(* IEC 61131-3 sources: xPLCCore/codesys_code/Application/APPs/AxisGroupSM (part 3) *)

(* ---- ProcessFlyEventsAndIo.st ---- *)
(* =========== IMPLEMENTATION =========== *)
// 2026-06-23 cleanup: trigger-arm + TTL boilerplate factored into
// ArmFiredTrigger() / TickTtl() helpers; pFly aliases the current slot
// once per iteration so the body reads `pFly^.X` instead of
// `FlyEventBuffer[Index].X` 20-odd times.
TriggerActive := FALSE;
FlyEventAvailableCount := 0;

FOR Index := 0 TO TO_INT(FlyEventBufferSize - 1) DO
    pFly := ADR(FlyEventBuffer[Index]);
    TriggerActive := FALSE;
    TriggerErrorCode := 0;

    CASE pFly^.TriggerType OF
        FlyEventTriggerType.DistanceTrigger:
            // Trigger by Cartesian distance from a fixed WCS point. Uses
            // squared distance to avoid SQRT on every scan. ReadPosition is
            // refreshed by UpdateAxisGroupState earlier in the same scan
            // (AxisGroupSM.st:346) so it's the actual TCP pose for this tick.
            DistDx := ReadPosition.c.x - pFly^.TargetPos_X;
            DistDy := ReadPosition.c.y - pFly^.TargetPos_Y;
            DistDz := ReadPosition.c.z - pFly^.TargetPos_Z;
            DistSq := DistDx*DistDx + DistDy*DistDy + DistDz*DistDz;
            DistThresholdSq := pFly^.TargetDistance * pFly^.TargetDistance;
            // TriggerInBoundary=TRUE: fire on entering the ball (dist <= radius).
            // TriggerInBoundary=FALSE: fire on leaving the ball (dist >= radius).
            IF (pFly^.TriggerInBoundary AND DistSq <= DistThresholdSq)
               OR (NOT pFly^.TriggerInBoundary AND DistSq >= DistThresholdSq) THEN
                TriggerActive := ArmFiredTrigger(pFly);
            ELSIF TickTtl(pFly) THEN
                TriggerActive := TRUE;
                TriggerErrorCode := TRIGGER_TIMEOUT_ERR;
            END_IF;

        FlyEventTriggerType.MovmentProgressTrigger:
            IF (
                CurrentMovementId > pFly^.TargetMovementId OR
                (CurrentMovementId = pFly^.TargetMovementId AND CurrentMovementIdProgress >= pFly^.TargetMovementProgress)
            ) THEN
                TriggerActive := ArmFiredTrigger(pFly);
            ELSIF TickTtl(pFly) THEN
                TriggerActive := TRUE;
                TriggerErrorCode := TRIGGER_TIMEOUT_ERR;
            END_IF;

        FlyEventTriggerType.PulseTrigger:
            // Phase 5: fire once GVL.ConveyorPulseRaw crosses the absolute
            // pulse target. Forward-only (>= test) -- a reset of the
            // conveyor encoder while events are pending will re-arm any
            // event with target <= current pulse, so producers must
            // re-issue M4s after a pulse-counter reset. TTL decay matches
            // DistanceTrigger / MovmentProgressTrigger semantics.
            IF (GVL.ConveyorPulseRaw >= pFly^.TargetPulseValue) THEN
                TriggerActive := ArmFiredTrigger(pFly);
            ELSIF TickTtl(pFly) THEN
                TriggerActive := TRUE;
                TriggerErrorCode := TRIGGER_TIMEOUT_ERR;
            END_IF;

        FlyEventTriggerType.SequenceDelayWait:
            IF (pFly^.IoStageIndex < pFly^.IoStageCount) THEN
                pFly^.IoStageDelayCountdown := pFly^.IoStageDelayCountdown - BusPeriod;
                IF (pFly^.IoStageDelayCountdown <= 0) THEN
                    TriggerActive := TRUE;
                END_IF;
            END_IF;

        FlyEventTriggerType.NOP:
            FlyEventAvailableCount := FlyEventAvailableCount + 1;
    END_CASE;

    IF (TriggerActive = FALSE) THEN
        CONTINUE;
    END_IF;

    IF (TriggerErrorCode <> 0) THEN
        // Drop-newest on overflow (see UpdateMotionProgress for SPSC race
        // rationale). The action-clear below still runs even if the error
        // event was dropped -- the FlyEvent itself is one-shot, not the
        // notification.
        IF (GVL.reMP_info_ridx.Space() > 0) THEN
            ResponsePacketPointer := ADR(GVL.reMP_info_arr[GVL.reMP_info_ridx.GetHead()]);
            MsgPakInfoClear(ResponsePacketPointer^);
            ResponsePacketPointer^.ele_count := ResponsePacketPointer^.ele_count + 3;

            ResponsePacketPointer^.whead := MessagePackerFb.PackString(pStart := ResponsePacketPointer^.whead, psValue := ADR('error_code'));
            ResponsePacketPointer^.whead := MessagePackerFb.PackDINT(pStart := ResponsePacketPointer^.whead, diValue := TriggerErrorCode);

            ResponsePacketPointer^.whead := MessagePackerFb.PackString(pStart := ResponsePacketPointer^.whead, psValue := ADR('src_id'));
            ResponsePacketPointer^.whead := MessagePackerFb.PackDINT(pStart := ResponsePacketPointer^.whead, diValue := pFly^.SourceCommandId);

            ResponsePacketPointer^.whead := MessagePackerFb.PackString(pStart := ResponsePacketPointer^.whead, psValue := ADR('event_id'));
            ResponsePacketPointer^.whead := MessagePackerFb.PackLINT(pStart := ResponsePacketPointer^.whead, liValue := TO_LINT(pFly^.EventId));

            MsgPakInfoWrapup(ResponsePacketPointer^);
            GVL.reMP_info_ridx.PushHead();
        ELSE
            GVL.ReMpDropCount := GVL.ReMpDropCount + 1;
            GVL.ReMpDropCount_TriggerEvent := GVL.ReMpDropCount_TriggerEvent + 1;
        END_IF;

        pFly^.ActionType := FlyEventActType.NOP;
        pFly^.TriggerType := FlyEventTriggerType.NOP;
    ELSE
        CASE pFly^.ActionType OF
            FlyEventActType.PIN_OPERATION:
                // Defensive bounds: guard against IoStageIndex >= IoStageCount
                // (post-increment lookup races) and against IoStageCount that
                // somehow exceeded FlyEventStageLimit (struct corruption).
                // Out-of-range deref of the fixed-size stage arrays would be
                // a hard crash; clamp to no-op instead.
                IF (pFly^.IoStageCount > 0
                    AND pFly^.IoStageIndex >= 0
                    AND pFly^.IoStageIndex < pFly^.IoStageCount
                    AND pFly^.IoStageIndex < FlyEventStageLimit) THEN
                    MotionOutputPin := pFly^.IoStagePinMask[pFly^.IoStageIndex];
                    StagePinState := pFly^.IoStagePinState[pFly^.IoStageIndex];
                ELSE
                    MotionOutputPin := 0;
                    StagePinState := 0;
                END_IF;

                TmpDigitalOutputBits := DigitalOutputBits;
                TmpDigitalOutputBits :=
                    (TmpDigitalOutputBits AND NOT (MotionOutputPin)) OR
                    ((StagePinState) AND (MotionOutputPin));
                DigitalOutputBits := TmpDigitalOutputBits;

                pFly^.IoStageIndex := pFly^.IoStageIndex + 1;
                IF (pFly^.IoStageIndex < pFly^.IoStageCount
                    AND pFly^.IoStageIndex < FlyEventStageLimit) THEN
                    pFly^.IoStageDelayCountdown := pFly^.IoStageDelay[pFly^.IoStageIndex];
                    pFly^.TriggerType := FlyEventTriggerType.SequenceDelayWait;
                ELSE
                    pFly^.ActionType := FlyEventActType.NOP;
                    pFly^.TriggerType := FlyEventTriggerType.NOP;
                END_IF;

                IoTriggerCount := IoTriggerCount + 1;

            FlyEventActType.COORD1_BIND:
                // Phase 4 step 3: apply the bind atomically when the
                // FlyEvent fires (typically via PulseTrigger at a precise
                // belt pulse). Belt is +X axis only for this phase, so
                // BindScaleY/Z are required to be 0 and BindScaleX != 0.
                // If we're already bound, this is a host-side sequencing
                // bug -> raise EV_ERROR with reason 'rebind_active' so
                // the operator sees a loud failure instead of a silent
                // wrong target.
                IF GVL.Coord1Bound THEN
                    // Latch the error context using the FlyEvent's own
                    // bookkeeping data so the host can correlate.
                    GVL.Coord1ErrPending     := TRUE;
                    GVL.Coord1ErrAtMovementId := CurrentMovementId;
                    GVL.Coord1ErrAtProgress  := CurrentMovementIdProgress;
                    GVL.Coord1ErrAtPulse     := GVL.ConveyorPulseRaw;
                    GVL.Coord1ErrAtArmX      := ReadPosition.c.x;
                    GVL.Coord1ErrAtArmY      := ReadPosition.c.y;
                    GVL.Coord1ErrAtArmZ      := ReadPosition.c.z;
                    GVL.Coord1ErrAtPcsX      := Pcs1KernelTransform.X;
                    GVL.Coord1ErrAtPcsY      := Pcs1KernelTransform.Y;
                    GVL.Coord1ErrAtPcsZ      := Pcs1KernelTransform.Z;
                    GVL.Coord1ErrRefPulse    := 0;  // bind never happened, no ref
                    GVL.Coord1ErrExitPulse   := GVL.Coord1ExitPulse;
                    GVL.Coord1BindEventId    := pFly^.EventId;
                    InputEvent := E_RobotEvent.EV_ERROR;
                ELSIF pFly^.BindScaleX = 0.0
                      OR pFly^.BindScaleY <> 0.0
                      OR pFly^.BindScaleZ <> 0.0 THEN
                    // Reject malformed bind -- same SM error path but with
                    // different latched event context for the host.
                    GVL.Coord1ErrPending     := TRUE;
                    GVL.Coord1ErrAtPulse     := GVL.ConveyorPulseRaw;
                    GVL.Coord1BindEventId    := pFly^.EventId;
                    InputEvent := E_RobotEvent.EV_ERROR;
                ELSE
                    // Trigger fire pulse used as ref_pulse so the bind is
                    // anchored at exactly the encoder value the host
                    // scheduled it for. PulseTrigger fires the same scan
                    // ConveyorPulseRaw first crosses TargetPulseValue, so
                    // current GVL.ConveyorPulseRaw is the right anchor.
                    Coord1PulseToMm := 1.0 / pFly^.BindScaleX;
                    Coord1BeltOriginRef.X := pFly^.BindRefXyzX
                                             - TO_LREAL(GVL.ConveyorPulseRaw) * Coord1PulseToMm;
                    Coord1BeltOriginRef.Y := pFly^.BindRefXyzY;
                    Coord1BeltOriginRef.Z := pFly^.BindRefXyzZ;
                    Coord1BeltOriginRef.A := 0.0;
                    Coord1BeltOriginRef.B := 0.0;
                    Coord1BeltOriginRef.C := 0.0;
                    GVL.Coord1RefPulse   := GVL.ConveyorPulseRaw;
                    GVL.Coord1RefXyz[0]  := pFly^.BindRefXyzX;
                    GVL.Coord1RefXyz[1]  := pFly^.BindRefXyzY;
                    GVL.Coord1RefXyz[2]  := pFly^.BindRefXyzZ;
                    GVL.Coord1Scale[0]   := pFly^.BindScaleX;
                    GVL.Coord1Scale[1]   := 0.0;
                    GVL.Coord1Scale[2]   := 0.0;
                    GVL.Coord1ExitPulse  := GVL.ConveyorPulseRaw
                                           + pFly^.BindExitPulseOffset;
                    GVL.Coord1BindEventId := pFly^.EventId;
                    GVL.Coord1CamMode    := GVL.COORD1_MODE_LINEAR;
                    GVL.Coord1CamCount   := 0;
                    GVL.Coord1Bound      := TRUE;
                    GVL.Coord1FlyBindActiveCount := GVL.Coord1FlyBindActiveCount + 1;
                END_IF;
                GVL.Coord1FlyBindCount := GVL.Coord1FlyBindCount + 1;
                pFly^.ActionType := FlyEventActType.NOP;
                pFly^.TriggerType := FlyEventTriggerType.NOP;

            FlyEventActType.ACK_SRC_ID://send ack with source command id
                // Drop-newest on overflow (SPSC race rationale in
                // UpdateMotionProgress). FlyEvent state is cleared either way
                // so we don't loop on the same one-shot.
                IF (GVL.reMP_info_ridx.Space() > 0) THEN
                    ResponsePacketPointer := ADR(GVL.reMP_info_arr[GVL.reMP_info_ridx.GetHead()]);
                    MsgPakInfoClear(ResponsePacketPointer^);

                    ResponsePacketPointer^.ele_count := ResponsePacketPointer^.ele_count +3;//three elements: event_id, id, ack

                    ResponsePacketPointer^.whead := MessagePackerFb.PackString(pStart := ResponsePacketPointer^.whead, psValue := ADR('event_id'));
                    ResponsePacketPointer^.whead := MessagePackerFb.PackLINT(pStart := ResponsePacketPointer^.whead, liValue := TO_LINT(pFly^.EventId));

                    ResponsePacketPointer^.whead := MessagePackerFb.PackString(pStart := ResponsePacketPointer^.whead, psValue := ADR('id'));
                    ResponsePacketPointer^.whead := MessagePackerFb.PackDINT(pStart := ResponsePacketPointer^.whead, diValue := pFly^.SourceCommandId);

                    ResponsePacketPointer^.whead := MessagePackerFb.PackString(pStart := ResponsePacketPointer^.whead, psValue := ADR('ack'));
                    ResponsePacketPointer^.whead := MessagePackerFb.PackBool(pStart := ResponsePacketPointer^.whead, bValue := TRUE);

                    MsgPakInfoWrapup(ResponsePacketPointer^);
                    GVL.reMP_info_ridx.PushHead();
                ELSE
                    GVL.ReMpDropCount := GVL.ReMpDropCount + 1;
                    GVL.ReMpDropCount_Reply := GVL.ReMpDropCount_Reply + 1;
                END_IF;

                pFly^.ActionType := FlyEventActType.NOP;
                pFly^.TriggerType := FlyEventTriggerType.NOP;

        END_CASE;
    END_IF;

    IoTriggerInfoCount := IoTriggerInfoCount + 1;
END_FOR;

//DigitalOutputPointer := IoConfig_Globals.HECAT_1616.OutputData;//////////////////////////////////////////////
OutputCHs[0] := TO_BYTE(DigitalOutputBits AND 16#FF);
OutputCHs[1] := TO_BYTE(SHR(DigitalOutputBits,8) AND 16#FF);

DBG_PIN:=0;
IF((DigitalOutputBits AND 16#4000)  >0)THEN
    DBG_PIN:=1;
END_IF
MoveLinearAbsoluteFb(
    AxisGroup := AxisGroupManagerFb._agAxisGroup,
    Execute := 0
);

GroupWaitFb(
    AxisGroup := AxisGroupManagerFb._agAxisGroup,
    Execute := 0
);

IF (RetryMotionCommandCooldown > 0) THEN
    RetryMotionCommandCooldown := RetryMotionCommandCooldown - BusPeriod;
END_IF;

// B1 diagnostic: latch the rising edge of Execute (=ApplyCoordTransform)
// BEFORE the FB call so we know exactly which scan kicked it off.
IF (ApplyCoordTransform AND NOT PrevApplyCoordTransform) THEN
    GVL.DBG_SetCoordExecuteRiseMs := RuntimeMs;
    DbgSetCoordSeenBusy  := FALSE;
    DbgSetCoordSeenDone  := FALSE;
    DbgSetCoordSeenError := FALSE;
END_IF;

SetCoordTransformFb(
    AxisGroup := AxisGroupManagerFb._agAxisGroup,
    Execute := ApplyCoordTransform,
    CoordTransform := CoordTransform,
    CoordSystem := SMC_COORD_SYSTEM.MCS
);

// B1 diagnostic: catch the FB lifecycle even if Busy is asserted for
// only a single scan. First-seen is what we care about; the FB clears
// Done/Error on the next falling-edge of Execute.
IF (SetCoordTransformFb.Busy AND NOT DbgSetCoordSeenBusy) THEN
    GVL.DBG_SetCoordBusyFirstMs := RuntimeMs;
    DbgSetCoordSeenBusy := TRUE;
END_IF;
IF (SetCoordTransformFb.Done AND NOT DbgSetCoordSeenDone) THEN
    GVL.DBG_SetCoordDoneMs := RuntimeMs;
    DbgSetCoordSeenDone := TRUE;
END_IF;
IF (SetCoordTransformFb.Error AND NOT DbgSetCoordSeenError) THEN
    GVL.DBG_SetCoordErrorMs := RuntimeMs;
    GVL.DBG_SetCoordLastErrorID := TO_DWORD(SetCoordTransformFb.ErrorID);
    DbgSetCoordSeenError := TRUE;
END_IF;

IF ApplyCoordTransform AND (SetCoordTransformFb.Busy OR SetCoordTransformFb.Done OR SetCoordTransformFb.Error) THEN
    ApplyCoordTransform := FALSE;
    GVL.DBG_SetCoordExecuteFallMs := RuntimeMs;
END_IF;
PrevApplyCoordTransform := ApplyCoordTransform;

ReadMcsTransformFb(
    AxisGroup := AxisGroupManagerFb._agAxisGroup,
    Enable := TRUE,
    CoordSystem := SMC_COORD_SYSTEM.MCS,
    Valid => ,
    Busy => ,
    Error => ,
    ErrorID => ,
    CoordTransform =>
);

// Phase 4 step 2 diagnostic: read kernel-side PCS_1 origin in WCS.
// MC_TrackConveyorBelt mutates this every scan; comparing it to the
// host-side prediction (GVL.Coord1OriginNow, formula-driven from
// RefXyz/RefPulse/Scale) confirms the FB is actually tracking the
// belt rather than holding a stale snapshot.
ReadPcs1TransformFb(
    AxisGroup := AxisGroupManagerFb._agAxisGroup,
    Enable := TRUE,
    CoordSystem := SMC_COORD_SYSTEM.PCS_1,
    Valid => ,
    Busy => ,
    Error => ,
    ErrorID => ,
    CoordTransform => Pcs1KernelTransform
);

(* ---- ProcessMotionPacket.st ---- *)
(* =========== IMPLEMENTATION =========== *)

    IF (RetryMotionCommandCooldown = 0 AND PacketType = 'M' AND GVL.minfo_buf_ridx.Size() > 0 AND MotionBufferSize < MOTION_BUFFER_THRESHOLD) THEN
        ShouldReturn := FALSE;
        CommandAck := FALSE;

        // reMP overflow guard: drop-newest. Producer must NOT ConsumeTail
        // (Comm task is sole consumer; two consumers race on _tail). When
        // the ring is full we route the pack into a scratch slot so the
        // long branchy block below can stay unchanged; PushHead at the
        // bottom is gated on SlotAvailable. See GVL.reMP_info_scratch.
        IF (GVL.reMP_info_ridx.Space() > 0) THEN
            SlotAvailable := TRUE;
            ResponsePacketPointer := ADR(GVL.reMP_info_arr[GVL.reMP_info_ridx.GetHead()]);
        ELSE
            SlotAvailable := FALSE;
            GVL.ReMpDropCount := GVL.ReMpDropCount + 1;
            GVL.ReMpDropCount_Reply := GVL.ReMpDropCount_Reply + 1;
            ResponsePacketPointer := ADR(GVL.reMP_info_scratch);
        END_IF;
        MsgPakInfoClear(ResponsePacketPointer^);
        MessagePackerFb.BindSlot(ResponsePacketPointer);  // builder pattern: pack helpers target this slot

        IF (GroupReadStatusFb.Error = TRUE OR GroupReadStatusFb.GroupErrorStop) THEN
            // Include an `err` string so the UI's NAK handler gets a readable
            // reason instead of the generic "nak (id=..., cmd=...)" fallback.
            IF (GroupReadStatusFb.GroupErrorStop) THEN
                MessagePackerFb.PackKvStr(ADR('err'), ADR('group_error_stop'));
            ELSE
                MessagePackerFb.PackKvStr(ADR('err'), ADR('group_read_status_error'));
            END_IF;
            MessagePackerFb.PackKvLint(ADR('ERROR_CODE'), GroupReadStatusFb.ErrorID);

            ShouldReturn := TRUE;
            CommandAck := FALSE;
            GVL.minfo_buf_ridx.ConsumeTail();

        ELSIF (CommandType = 'BLOCK_FOR_MOTION_STOP' OR CommandType = 'WAIT_FOR_MOTION_STOP'
               OR CommandType = 'WAIT_FOR_REEL_STOP' OR CommandType = 'BLOCK_FOR_REEL_STOP'
               OR CommandType = 'BLOCK_FOR_DIGITAL_INPUT') THEN
            // Deferred-reply waits (review 2026-09-24 P0-3). Registered and
            // taken off the queue at once; the main body (pending waits
            // block) acks when the condition holds, NAKs block_timeout on
            // expiry or group_not_ready when the FSM leaves Ready. Packets
            // behind a wait are no longer held: a wait is not a barrier.
            // One pending wait per kind; a second one NAKs wait_busy.
            IF (CommandType = 'BLOCK_FOR_DIGITAL_INPUT') THEN
                WaitKind := WAIT_KIND_DIN;
            ELSIF (CommandType = 'WAIT_FOR_REEL_STOP' OR CommandType = 'BLOCK_FOR_REEL_STOP') THEN
                WaitKind := WAIT_KIND_REEL;
            ELSE
                WaitKind := WAIT_KIND_MOTION;
            END_IF;

            IF WaitActive[WaitKind] THEN
                MessagePackerFb.PackKvStr(ADR('err'), ADR('wait_busy'));
                ShouldReturn := TRUE;
                CommandAck := FALSE;
            ELSIF (WaitKind = WAIT_KIND_DIN)
                  AND (MessageUnpackerFb.TryReadINT64('group', 0) < 0
                       OR MessageUnpackerFb.TryReadINT64('group', 0) > 1) THEN
                // DigitalInputPointer[group] reads 2 bytes (SimDigitalInput
                // / InputCHs); a larger host index read past them.
                MessagePackerFb.PackKvStr(ADR('err'), ADR('bad_group'));
                ShouldReturn := TRUE;
                CommandAck := FALSE;
            ELSE
                WaitActive[WaitKind]    := TRUE;
                WaitCmdId[WaitKind]     := CommandId;
                WaitStartMs[WaitKind]   := RuntimeMs;
                WaitTimeoutMs[WaitKind] := MessageUnpackerFb.TryReadINT64('timeout_ms', 0);
                IF (WaitKind = WAIT_KIND_DIN) THEN
                    WaitPinMask  := TO_UINT(MessageUnpackerFb.TryReadINT64('pin', 0));
                    WaitPinGroup := TO_UINT(MessageUnpackerFb.TryReadINT64('group', 0));
                    WaitPinState := TO_UINT(MessageUnpackerFb.TryReadINT64('state', 0));
                    // "Wait forever" on an input is how the PLC wedged
                    // before; inputs get a ceiling instead.
                    IF (WaitTimeoutMs[WaitKind] <= 0) THEN
                        WaitTimeoutMs[WaitKind] := WAIT_DIN_DEFAULT_TIMEOUT_MS;
                    END_IF;
                END_IF;
                // No reply now: it is sent when the wait resolves.
            END_IF;
            GVL.minfo_buf_ridx.ConsumeTail();

        ELSIF (CommandType = 'GET_DIGITAL_INPUT') THEN
            //InputPinGroup := TO_UINT(MessageUnpackerFb.TryReadINT64('group', 0));

            IF DigitalInputPointer <> 0 THEN
                MessagePackerFb.PackKvDint(ADR('state'), DigitalInputPointer[0] OR SHL(TO_UDINT(DigitalInputPointer[1]), 8));
            ELSE
                // DigitalInputPointer not wired (HECAT_1616 line in TrackDigitalInputFlips is commented out).
                // Return 0 rather than dereferencing null.
                MessagePackerFb.PackKvDint(ADR('state'), 0);
            END_IF;

            ShouldReturn := TRUE;
            CommandAck := TRUE;
            GVL.minfo_buf_ridx.ConsumeTail();
        ELSIF (CommandType = 'READ_LATEST_CMD_LOCATION') THEN

            MessagePackerFb.PackKvReal(ADR('X'), TO_REAL(MotionPose.c.X));
            MessagePackerFb.PackKvReal(ADR('Y'), TO_REAL(MotionPose.c.Y));
            MessagePackerFb.PackKvReal(ADR('Z'), TO_REAL(MotionPose.c.Z));
            MessagePackerFb.PackKvReal(ADR('A'), TO_REAL(G1ADeg));   // degrees, as sent in G1
            MessagePackerFb.PackKvReal(ADR('B'), TO_REAL(MotionPose.c.B));
            MessagePackerFb.PackKvReal(ADR('C'), TO_REAL(MotionPose.c.C));

            ShouldReturn := TRUE;
            CommandAck := TRUE;
            GVL.minfo_buf_ridx.ConsumeTail();

        ELSIF (CommandType = 'G4') THEN
            // B1 fix (analysis 1.5, test_plc_refactor_findings_b2): do NOT
            // set ShouldReturn/CommandAck at branch entry. Pre-fix they were
            // set here, BEFORE SMC_GroupWait ran -- on CommandAccepted=FALSE
            // the packet stayed queued but the tail-commit still emitted
            // ack:TRUE (without movement_id), then every 100ms retry
            // cooldown re-acked the same id. Mirror the G1 branch: reply
            // only from the accepted / NAK paths.
            G4HaltTime := MessageUnpackerFb.TryReadREAL('P', - 1);

            IF (G4HaltTime > 0) THEN
                GroupWaitFb(
                    AxisGroup := AxisGroupManagerFb._agAxisGroup,
                    Execute := 1,
                    WaitTime := G4HaltTime
                );

                IF (GroupWaitFb.CommandAccepted) THEN
                    GVL.minfo_buf_ridx.ConsumeTail();

                    MessagePackerFb.PackKvLint(ADR('movement_id'), TO_LINT(GroupWaitFb.MovementId));

                    ShouldReturn := TRUE;
                    CommandAck := TRUE;
                ELSE
                    RetryMotionCommandCooldown := RETRY_COOLDOWN_G4_MS;
                END_IF;
            ELSE
                // P <= 0 (or missing): NAK with a reason (R2 spirit --
                // no bare NAKs).
                MessagePackerFb.PackKvStr(ADR('err'), ADR('bad_dwell'));
                GVL.minfo_buf_ridx.ConsumeTail();

                ShouldReturn := TRUE;
                CommandAck := FALSE;
            END_IF;

        ELSIF (CommandType = 'SetCoord0') THEN
            // 2026-06-23 code-review fix: refuse if a G1 is in flight.
            // Pulsing MC_SetCoordinateTransform while a move is executing
            // shifts the WCS origin under the move and the arm darts.
            // Mirrors COORD1_BIND's own motion-in-flight guard.
            IF MotionBufferSize > 0 THEN
                MessagePackerFb.PackKvStr(ADR('err'), ADR('motion_in_flight'));
                GVL.SetCoordBusyNakCount := GVL.SetCoordBusyNakCount + 1;
                ShouldReturn := TRUE;
                CommandAck := FALSE;
                GVL.minfo_buf_ridx.ConsumeTail();
            ELSE
                CoordTransform.X := 0.0;
                CoordTransform.Y := 0.0;
                CoordTransform.Z := 0.0;
                CoordTransform.A := 0.0;
                CoordTransform.B := 0.0;
                CoordTransform.C := 0.0;
                ApplyCoordTransform := TRUE;
                GVL.CoordSystemConfigured := TRUE;

                ShouldReturn := TRUE;
                CommandAck := TRUE;
                GVL.minfo_buf_ridx.ConsumeTail();
            END_IF

        ELSIF (CommandType = 'SetCoord1') THEN
            // Same guard as SetCoord0 -- see comment above.
            IF MotionBufferSize > 0 THEN
                MessagePackerFb.PackKvStr(ADR('err'), ADR('motion_in_flight'));
                GVL.SetCoordBusyNakCount := GVL.SetCoordBusyNakCount + 1;
                ShouldReturn := TRUE;
                CommandAck := FALSE;
                GVL.minfo_buf_ridx.ConsumeTail();
            ELSE
                CoordTransform.X := 0.0;
                CoordTransform.Y := 0.0;
                CoordTransform.Z := 0.0;
                CoordTransform.A := COORD1_FRAME_A;
                CoordTransform.B := 0.0;
                CoordTransform.C := 0.0;
                ApplyCoordTransform := TRUE;
                GVL.CoordSystemConfigured := TRUE;
                GVL.DBG_SetCoord1AcceptMs := RuntimeMs;
                // Reset the lifecycle DBG_SetCoord* fields so an old reading
                // doesn't get mistaken for the new run.
                GVL.DBG_SetCoordExecuteRiseMs  := 0;
                GVL.DBG_SetCoordBusyFirstMs    := 0;
                GVL.DBG_SetCoordDoneMs         := 0;
                GVL.DBG_SetCoordErrorMs        := 0;
                GVL.DBG_SetCoordLastErrorID    := 0;
                GVL.DBG_SetCoordExecuteFallMs  := 0;

                ShouldReturn := TRUE;
                CommandAck := TRUE;
                GVL.minfo_buf_ridx.ConsumeTail();
            END_IF

        ELSIF (CommandType = 'RESET_DBG_INFO') THEN
            // Legacy M-path branch (wire-visible; some old callers use it).
            // R8 fix: delegate to the ONE canonical list so the two paths
            // can never drift again.
            ResetDiagCounters();
            ShouldReturn := TRUE;
            CommandAck := TRUE;
            GVL.minfo_buf_ridx.ConsumeTail();

        ELSIF (CommandType = 'TAPE_CYCLE') THEN
            // Tape step as one command (plc.md §Direction step 3): when the
            // move motion_id_offset / motion_progress relative to the last
            // accepted one starts, advance the reel by Distance (0 = none)
            // and wait for it, then arm the pin_op_seq shots as a
            // DistanceTrigger fly event (fire once the arm is outside the
            // sphere tx/ty/tz/td). Deferred reply {wait_ms, reel_ms} when
            // the shots are armed; NAK tape_busy / flyevent_buffer_full /
            // tape_timeout / reel_busy / group_not_ready. See the TAPE_CYCLE
            // block in AxisGroupSM.
            IF TapeActive OR ReelTrkActive THEN
                MessagePackerFb.PackKvStr(ADR('err'), ADR('tape_busy'));
                ShouldReturn := TRUE;
                CommandAck := FALSE;
            ELSIF GVL.ReelMvOpen THEN
                // a fault stopped the last tape move short: the tape is
                // between cells until REEL_RESUME / REEL_CLEAR
                MessagePackerFb.PackKvStr(ADR('err'), ADR('reel_interrupted'));
                ShouldReturn := TRUE;
                CommandAck := FALSE;
            ELSIF (FlyEventAvailableCount <= 3) THEN
                MessagePackerFb.PackKvStr(ADR('err'), ADR('flyevent_buffer_full'));
                ShouldReturn := TRUE;
                CommandAck := FALSE;
            ELSE
                TapeTargetId := GroupReadStatusFb.LastAcceptedMovementId;
                TapeOffset := TO_DINT(MessageUnpackerFb.TryReadINT64('motion_id_offset', 0));
                IF TapeOffset >= 0 THEN
                    TapeTargetId := TapeTargetId + DINT_TO_ULINT(TapeOffset);
                ELSIF TapeTargetId >= DINT_TO_ULINT(-TapeOffset) THEN
                    TapeTargetId := TapeTargetId - DINT_TO_ULINT(-TapeOffset);
                ELSE
                    TapeTargetId := 0;
                END_IF;
                TapeTargetProg := MessageUnpackerFb.TryReadREAL('motion_progress', 0);
                TapeReelDist := MessageUnpackerFb.TryReadREAL('Distance', 0);
                TapeReelF    := MessageUnpackerFb.TryReadREAL('F',    reelGoVelocity);
                TapeReelAcc  := MessageUnpackerFb.TryReadREAL('ACC',  reelGoAccel);
                TapeReelDec  := MessageUnpackerFb.TryReadREAL('DEA',  reelGoDecel);
                TapeReelJerk := MessageUnpackerFb.TryReadREAL('JERK', reelGoJerk);
                TapeTimeoutMs := MessageUnpackerFb.TryReadINT64('timeout_ms', 0);
                // Plan tracking: cells this step advances, added to
                // GVL.PlanCellsDone once the reel has actually moved.
                TapePlanCells := TO_DINT(MessageUnpackerFb.TryReadINT64('cells', 0));
                TapePlanKind  := TO_INT(MessageUnpackerFb.TryReadINT64('kind', 0));
                IF TapeTimeoutMs <= 0 THEN
                    TapeTimeoutMs := TAPE_DEFAULT_TIMEOUT_MS;
                END_IF;

                // the shots: a DistanceTrigger pin op, as M4 trig 120 builds it
                TapeFly.ActionType := FlyEventActType.PIN_OPERATION;
                TapeFly.TriggerType := FlyEventTriggerType.DistanceTrigger;
                TapeFly.SourceCommandId := CommandId;
                TapeFly.PinGrp := 0;
                TapeFly.TimeToLiveMs := TO_DINT(MessageUnpackerFb.TryReadINT64('ttl_ms', 3000));
                TapeFly.TargetMovementId := 0;
                TapeFly.TargetMovementProgress := 0;
                TapeFly.TargetPos_X := TO_LREAL(MessageUnpackerFb.TryReadREAL('tx', 0));
                TapeFly.TargetPos_Y := TO_LREAL(MessageUnpackerFb.TryReadREAL('ty', 0));
                TapeFly.TargetPos_Z := TO_LREAL(MessageUnpackerFb.TryReadREAL('tz', 0));
                TapeFly.TargetDistance := TO_LREAL(MessageUnpackerFb.TryReadREAL('td', 0));
                TapeFly.TriggerInBoundary := MessageUnpackerFb.TryReadINT64('tin', 0) <> 0;
                TapeFly.TargetPulseValue := 0;
                TapeFly.EventId := TO_DINT(MessageUnpackerFb.TryReadINT64('event_id', 0));
                TapeFly.IoStageCount := 0;
                TapeFly.IoStageIndex := 0;
                TapeFly.IoStageDelayCountdown := 0;
                FOR StageLoopIdx := 0 TO FlyEventStageLimit-1 DO
                    TapeFly.IoStageDelay[StageLoopIdx] := 0;
                    TapeFly.IoStagePinMask[StageLoopIdx] := 0;
                    TapeFly.IoStagePinState[StageLoopIdx] := 0;
                END_FOR;
                IF MessageUnpackerFb.TryReadObject('pin_op_seq', ADR(fbPinOpSeqUnpacker)) THEN
                    fbPinOpSeqUnpacker.UnpackNext();
                    FOR PinOpSeqIdx := 0 TO (fbPinOpSeqUnpacker.uiLastCount / 3) - 1 DO
                        IF TapeFly.IoStageCount >= FlyEventStageLimit THEN
                            EXIT;
                        END_IF;
                        fbPinOpSeqUnpacker.UnpackNext();
                        StageDelayTemp := LIMIT(0, fbPinOpSeqUnpacker.diLastDINT, 600000);  // ms; TO_INT wrapped past 32767
                        fbPinOpSeqUnpacker.UnpackNext();
                        IF fbPinOpSeqUnpacker.diLastDINT < 0 THEN StagePinMaskTemp := 0;
                        ELSE StagePinMaskTemp := DINT_TO_ULINT(fbPinOpSeqUnpacker.diLastDINT); END_IF;
                        fbPinOpSeqUnpacker.UnpackNext();
                        IF fbPinOpSeqUnpacker.diLastDINT < 0 THEN StagePinStateTemp := 0;
                        ELSE StagePinStateTemp := DINT_TO_ULINT(fbPinOpSeqUnpacker.diLastDINT); END_IF;
                        IF StagePinMaskTemp <> 0 THEN
                            TapeFly.IoStageDelay[TapeFly.IoStageCount] := StageDelayTemp;
                            TapeFly.IoStagePinMask[TapeFly.IoStageCount] := StagePinMaskTemp;
                            TapeFly.IoStagePinState[TapeFly.IoStageCount] := StagePinStateTemp;
                            TapeFly.IoStageCount := TapeFly.IoStageCount + 1;
                        END_IF;
                    END_FOR;
                END_IF;

                // Reserve the shots' slot now, before the reel moves, so a
                // full buffer is refused here instead of after the advance.
                TapeSlotIdx := -1;
                FOR TapeIdx := 0 TO TO_INT(FlyEventBufferSize - 1) DO
                    IF FlyEventBuffer[TapeIdx].TriggerType = FlyEventTriggerType.NOP THEN
                        FlyEventBuffer[TapeIdx].TriggerType := FlyEventTriggerType.Reserved;
                        TapeSlotIdx := TapeIdx;
                        EXIT;
                    END_IF;
                END_FOR;
                IF TapeSlotIdx < 0 THEN
                    MessagePackerFb.PackKvStr(ADR('err'), ADR('flyevent_buffer_full'));
                    ShouldReturn := TRUE;
                    CommandAck := FALSE;
                ELSE
                    TapeCmdId := CommandId;
                    TapeStartMs := RuntimeMs;
                    TapeState := 1;
                    TapeActive := TRUE;
                    // no reply now: it comes when the shots are armed
                END_IF;
            END_IF;
            GVL.minfo_buf_ridx.ConsumeTail();

        ELSIF (CommandType = 'ReelGo') THEN
            // NAK instead of acking a move that will not happen: while a
            // TAPE_CYCLE owns the reel (it moves through the same reelGo*
            // parameters, which this would overwrite), or when both FB
            // instances are busy (active + queued). Both used to ack TRUE.
            IF TapeActive OR ReelTrkActive THEN
                MessagePackerFb.PackKvStr(ADR('err'), ADR('tape_busy'));
                CommandAck := FALSE;
            ELSIF reelMoveRelative.Busy AND reelMoveRelative2.Busy THEN
                MessagePackerFb.PackKvStr(ADR('err'), ADR('reel_busy'));
                CommandAck := FALSE;
            ELSE
                reelGoDistance := MessageUnpackerFb.TryReadREAL('Distance', reelGoDistance);
                reelGoVelocity := MessageUnpackerFb.TryReadREAL('F',        reelGoVelocity);
                reelGoAccel    := MessageUnpackerFb.TryReadREAL('ACC',      reelGoAccel);
                reelGoDecel    := MessageUnpackerFb.TryReadREAL('DEA',      reelGoDecel);
                reelGoJerk     := MessageUnpackerFb.TryReadREAL('JERK',     reelGoJerk);
                IF NOT reelMoveRelative.Busy THEN
                    reelGoRequest  := TRUE;
                ELSE
                    reelGoRequest2 := TRUE;
                END_IF;
                CommandAck := TRUE;
            END_IF;
            ShouldReturn := TRUE;
            GVL.minfo_buf_ridx.ConsumeTail();

        ELSIF (CommandType = 'M4') THEN

				MotionTargetMovementId := TO_ULINT(MessageUnpackerFb.TryReadUINT64('motion_id', TO_ULINT(GroupReadStatusFb.LastAcceptedMovementId)));

				MessagePackerFb.PackKvLint(ADR('ev_buf_space'), TO_LINT(FlyEventAvailableCount));

				IF (FlyEventAvailableCount > 3) THEN

					// Phase 4 step 3: 'action' field switches between pin
					// operation (default, legacy) and scheduled COORD1_BIND.
					FlyEventTempData := FlyEventBlank;
					M4ActionStr := MessageUnpackerFb.TryReadString('action', 'pin_op');
					IF M4ActionStr = 'coord1_bind' THEN
						FlyEventTempData.ActionType := FlyEventActType.COORD1_BIND;
					ELSE
						FlyEventTempData.ActionType := FlyEventActType.PIN_OPERATION;
					END_IF;

					// Optional 'trig' field selects trigger family. Default
					// 20 = MovmentProgressTrigger preserves legacy callers
					// that omit the field. 120 = DistanceTrigger uses a
					// Cartesian point + radius gate instead of motion_id.
					// 130 = PulseTrigger gates on GVL.ConveyorPulseRaw
					// threshold (Phase 5: conveyor pick).
					FlyEventTriggerSelect := TO_INT(MessageUnpackerFb.TryReadINT64('trig', 20));
					IF FlyEventTriggerSelect = 120 THEN
						FlyEventTempData.TriggerType := FlyEventTriggerType.DistanceTrigger;
					ELSIF FlyEventTriggerSelect = 130 THEN
						FlyEventTempData.TriggerType := FlyEventTriggerType.PulseTrigger;
					ELSE
						FlyEventTempData.TriggerType := FlyEventTriggerType.MovmentProgressTrigger;
					END_IF;

					FlyEventTempData.SourceCommandId := CommandId;

					FlyEventTempData.PinGrp := 0;

					// 2026-06-23: legacy 'reset_ms' wire field removed. Hosts now
					// pass the equivalent 2-stage sequence via pin_op_seq (handled
					// below). lib/protocol.ts cmd.M4 keeps the `reset_ms:N` host
					// API alive by expanding to pin_op_seq client-side, so TS call
					// sites don't change; python tests use tests/_raw_plc.m4_pulse_seq.

					FlyEventTtlRaw := MessageUnpackerFb.TryReadINT64('ttl_ms', -1);
					IF (FlyEventTtlRaw < 0) OR (FlyEventTtlRaw > 2147483647) THEN
						FlyEventTempData.TimeToLiveMs := -1;
					ELSE
						FlyEventTempData.TimeToLiveMs := TO_DINT(FlyEventTtlRaw);
					END_IF;

					// Read offset as full DINT (was TO_INT, which silently wrapped
					// any value >32767 to negative and rolled TargetMovementId
					// backwards onto a stale movement). Negative offsets that
					// would underflow ULINT are clamped to 0.
					MotionIdOffsetTemp := TO_DINT(MessageUnpackerFb.TryReadINT64('motion_id_offset', 0));
					IF MotionIdOffsetTemp >= 0 THEN
						FlyEventTempData.TargetMovementId := MotionTargetMovementId + DINT_TO_ULINT(MotionIdOffsetTemp);
					ELSIF MotionTargetMovementId >= DINT_TO_ULINT(-MotionIdOffsetTemp) THEN
						FlyEventTempData.TargetMovementId := MotionTargetMovementId - DINT_TO_ULINT(-MotionIdOffsetTemp);
					ELSE
						FlyEventTempData.TargetMovementId := 0;
					END_IF;

					FlyEventTempData.TargetMovementProgress := TO_LREAL(MessageUnpackerFb.TryReadREAL('motion_progress', 1));

					// DistanceTrigger payload (ignored by MovmentProgressTrigger).
					// Defaults to (0,0,0)/r=0/inside; with r=0 and TriggerInBoundary=TRUE
					// the trigger fires only at the exact origin -- safe default that
					// just won't fire on its own. tin: 0=outside, 1=inside.
					FlyEventTempData.TargetPos_X := TO_LREAL(MessageUnpackerFb.TryReadREAL('tx', 0));
					FlyEventTempData.TargetPos_Y := TO_LREAL(MessageUnpackerFb.TryReadREAL('ty', 0));
					FlyEventTempData.TargetPos_Z := TO_LREAL(MessageUnpackerFb.TryReadREAL('tz', 0));
					FlyEventTempData.TargetDistance := TO_LREAL(MessageUnpackerFb.TryReadREAL('td', 0));
					FlyEventTempData.TriggerInBoundary := MessageUnpackerFb.TryReadINT64('tin', 1) <> 0;

					// PulseTrigger payload (ignored by other trigger types). Default
					// 0 means "fire immediately on next scan if ConveyorPulseRaw>=0",
					// which for an idle conveyor (Pulse=0) and a forgotten field is
					// safe-ish only with a positive TTL. Callers should supply an
					// explicit pulse target.
					FlyEventTempData.TargetPulseValue := TO_DINT(MessageUnpackerFb.TryReadINT64('pulse_target', 0));

					// COORD1_BIND action payload (Phase 4 step 3). Only meaningful
					// when ActionType = COORD1_BIND; other actions ignore. Pulled
					// off the wire unconditionally to keep the parser simple --
					// stale reads cost a handful of cycles, not correctness.
					FlyEventTempData.BindRefXyzX := TO_LREAL(MessageUnpackerFb.TryReadREAL('ref_xyz[0]', 0));
					FlyEventTempData.BindRefXyzY := TO_LREAL(MessageUnpackerFb.TryReadREAL('ref_xyz[1]', 0));
					FlyEventTempData.BindRefXyzZ := TO_LREAL(MessageUnpackerFb.TryReadREAL('ref_xyz[2]', 0));
					FlyEventTempData.BindScaleX  := TO_LREAL(MessageUnpackerFb.TryReadREAL('scale[0]', 0));
					FlyEventTempData.BindScaleY  := TO_LREAL(MessageUnpackerFb.TryReadREAL('scale[1]', 0));
					FlyEventTempData.BindScaleZ  := TO_LREAL(MessageUnpackerFb.TryReadREAL('scale[2]', 0));
					FlyEventTempData.BindExitPulseOffset := TO_DINT(MessageUnpackerFb.TryReadINT64('exit_pulse_offset', 0));

					FlyEventTempData.EventId := TO_DINT(MessageUnpackerFb.TryReadINT64('event_id', 0));

					FlyEventTempData.IoStageCount := 0;

					FlyEventTempData.IoStageIndex := 0;

					FlyEventTempData.IoStageDelayCountdown := 0;

					FOR StageLoopIdx := 0 TO FlyEventStageLimit-1 DO

						FlyEventTempData.IoStageDelay[StageLoopIdx] := 0;

						FlyEventTempData.IoStagePinMask[StageLoopIdx] := 0;

						FlyEventTempData.IoStagePinState[StageLoopIdx] := 0;

					END_FOR;

					(* Parse pin_op_seq array: [delay0, pin0, state0, delay1, pin1, state1, ...] *)
					(* Use sequential reading with array unpacker for fast performance - no string operations *)
					IF MessageUnpackerFb.TryReadObject('pin_op_seq', ADR(fbPinOpSeqUnpacker)) THEN
						(* Read array header to get length *)
						fbPinOpSeqUnpacker.UnpackNext();

						(* Loop through array in groups of 3 (delay, pin, state) *)
						FOR PinOpSeqIdx := 0 TO (fbPinOpSeqUnpacker.uiLastCount / 3) - 1 DO
							IF FlyEventTempData.IoStageCount >= FlyEventStageLimit THEN
								EXIT; (* Reached maximum stage limit *)
							END_IF;

							(* Read delay value (signed integer) - sequential read *)
							fbPinOpSeqUnpacker.UnpackNext();
							StageDelayTemp := LIMIT(0, fbPinOpSeqUnpacker.diLastDINT, 600000);  // ms; TO_INT wrapped past 32767

							(* Read pin mask value (unsigned integer) - sequential read *)
							(* UnpackNext reads integers into diLastDINT; convert to ULINT for unsigned values *)
							fbPinOpSeqUnpacker.UnpackNext();
							(* Pin masks are bit patterns, inherently non-negative. Clamp negative
							   DINT values (e.g. client sent a signed negative int by mistake) to 0
							   so we don't wrap into a huge ULINT and trigger unintended outputs. *)
							IF fbPinOpSeqUnpacker.diLastDINT < 0 THEN
								StagePinMaskTemp := 0;
							ELSE
								StagePinMaskTemp := DINT_TO_ULINT(fbPinOpSeqUnpacker.diLastDINT);
							END_IF;

							(* Read pin state value (unsigned integer) - sequential read *)
							fbPinOpSeqUnpacker.UnpackNext();
							IF fbPinOpSeqUnpacker.diLastDINT < 0 THEN
								StagePinStateTemp := 0;
							ELSE
								StagePinStateTemp := DINT_TO_ULINT(fbPinOpSeqUnpacker.diLastDINT);
							END_IF;

							(* Only add stage if pin mask is non-zero *)
							IF StagePinMaskTemp <> 0 THEN
								FlyEventTempData.IoStageDelay[FlyEventTempData.IoStageCount] := StageDelayTemp;
								FlyEventTempData.IoStagePinMask[FlyEventTempData.IoStageCount] := StagePinMaskTemp;
								FlyEventTempData.IoStagePinState[FlyEventTempData.IoStageCount] := StagePinStateTemp;
								FlyEventTempData.IoStageCount := FlyEventTempData.IoStageCount + 1;
							END_IF;
						END_FOR;
					END_IF;

					// 2026-06-23: legacy `{pin, state, reset_ms}` single-pulse shape
					// removed. This block previously auto-appended one stage from
					// `pin` + `state` plus an optional reset stage from `ResetDelayMs`.
					// Both moved client-side (lib/protocol.ts expandM4ResetMs +
					// tests/_raw_plc.m4_pulse_seq) so the PLC has a single canonical
					// input: pin_op_seq.

					// Registration gate: progress trigger needs a real target movement id;
					// distance + pulse triggers don't (they gate on Cartesian pose /
					// conveyor pulse), so accept regardless of MotionTargetMovementId
					// for those branches. COORD1_BIND action has no IO stages and
					// MUST be paired with PulseTrigger (gates the bind on a precise
					// conveyor pulse); refuse the registration otherwise so a host
					// can't accidentally end up with a never-firing bind sitting in
					// the slot.
					IF (FlyEventTempData.ActionType = FlyEventActType.COORD1_BIND
					    AND FlyEventTempData.TriggerType = FlyEventTriggerType.PulseTrigger
					    AND FlyEventTempData.BindExitPulseOffset > 0)
					   OR (FlyEventTempData.ActionType = FlyEventActType.PIN_OPERATION
					       AND FlyEventTempData.IoStageCount > 0
					       AND (MotionTargetMovementId <> 0
					            OR FlyEventTempData.TriggerType = FlyEventTriggerType.DistanceTrigger
					            OR FlyEventTempData.TriggerType = FlyEventTriggerType.PulseTrigger)) THEN

						FOR Index := 0 TO TO_INT( FlyEventBufferSize - 1) DO

							IF (FlyEventBuffer[Index].TriggerType = 0) THEN

								FlyEventBuffer[Index] := FlyEventTempData;

								CommandAck := TRUE;

								EXIT;

							END_IF;

						END_FOR;

						IoCommandCount := IoCommandCount + 1;

						ShouldReturn := TRUE;

					ELSE
						// R3/R4 fix (test_plc_refactor_findings): a rejected
						// registration used to be consumed with no reply and
						// no counter -- a no_silent_drops violation the host
						// could only see as a timeout. NAK with the reason.
						ShouldReturn := TRUE;
						CommandAck := FALSE;
						MessagePackerFb.PackKvStr(ADR('err'), ADR('flyevent_reject'));
						GVL.FlyEventRejectNakCount := GVL.FlyEventRejectNakCount + 1;
					END_IF;

					GVL.minfo_buf_ridx.ConsumeTail();

				ELSE
					// R11 fix: with <=3 free slots the M4 used to sit
					// unconsumed at the minfo tail; the dispatcher EXITs on a
					// type-M tail, so EVERY packet behind it (SYS included)
					// stalled with zero counters -- an invisible full-queue
					// wedge. NAK + consume keeps the queue draining; the
					// packet is retryable by the host once slots free up.
					ShouldReturn := TRUE;
					CommandAck := FALSE;
					MessagePackerFb.PackKvStr(ADR('err'), ADR('flyevent_buffer_full'));
					GVL.FlyEventBufferFullNakCount := GVL.FlyEventBufferFullNakCount + 1;
					GVL.minfo_buf_ridx.ConsumeTail();

				END_IF;

ELSIF (CommandType = 'WAIT_FOR_TRIGGER_MOTION_PROGRESS') THEN
            IF (FlyEventAvailableCount > 3) THEN

                MotionTargetMovementId := TO_ULINT(MessageUnpackerFb.TryReadINT64('motion_id', TO_LINT(GroupReadStatusFb.LastAcceptedMovementId)));

                // R5 fix: the old gate also required MotionOutputPin <> 0 --
                // a copy-paste leftover from the legacy M4 shape.
                // MotionOutputPin is ProcessFlyEventsAndIo's scratch (the pin
                // mask of the LAST FIRED pin-op stage), semantically unrelated
                // to this registration; until any pin-op ever fired it is 0
                // and every registration was refused -- silently (see ELSE).
                IF (MotionTargetMovementId <> 0) THEN
                    // It set only the fields below and inherited the rest --
                    // pin stages, delays, sphere -- from the last M4.
                    FlyEventTempData := FlyEventBlank;
                    FlyEventTempData.ActionType := FlyEventActType.ACK_SRC_ID;
                    FlyEventTempData.TriggerType := FlyEventTriggerType.MovmentProgressTrigger;
                    // Same TO_INT->INT16 wrap fix as the M4 branch above.
                    MotionIdOffsetTemp := TO_DINT(MessageUnpackerFb.TryReadINT64('motion_id_offset', 0));
                    IF MotionIdOffsetTemp >= 0 THEN
                        FlyEventTempData.TargetMovementId := MotionTargetMovementId + DINT_TO_ULINT(MotionIdOffsetTemp);
                    ELSIF MotionTargetMovementId >= DINT_TO_ULINT(-MotionIdOffsetTemp) THEN
                        FlyEventTempData.TargetMovementId := MotionTargetMovementId - DINT_TO_ULINT(-MotionIdOffsetTemp);
                    ELSE
                        FlyEventTempData.TargetMovementId := 0;
                    END_IF;
                    FlyEventTempData.TargetMovementProgress := TO_LREAL(MessageUnpackerFb.TryReadREAL('motion_progress', 1));

                    FlyEventTempData.SourceCommandId := CommandId;

                    FlyEventTempData.EventId := TO_DINT(MessageUnpackerFb.TryReadINT64('event_id', 0));
                    FlyEventTtlRaw := MessageUnpackerFb.TryReadINT64('ttl_ms', -1);
                    IF (FlyEventTtlRaw < 0) OR (FlyEventTtlRaw > 2147483647) THEN
                        FlyEventTempData.TimeToLiveMs := -1;
                    ELSE
                        FlyEventTempData.TimeToLiveMs := TO_DINT(FlyEventTtlRaw);
                    END_IF;

                    FOR Index := 0 TO TO_INT(FlyEventBufferSize - 1) DO
                        IF (FlyEventBuffer[Index].TriggerType = 0) THEN
                            FlyEventBuffer[Index] := FlyEventTempData;
                            EXIT;
                        END_IF;
                    END_FOR;
                    // Registration OK: no immediate reply -- the ack is
                    // deferred and arrives as the ACK_SRC_ID event when the
                    // trigger fires (ShouldReturn deliberately stays FALSE).
                ELSE
                    // R5 fix: refusal used to consume the packet with
                    // ShouldReturn never set -> host timed out with nothing
                    // in any counter. NAK like every other reject path.
                    ShouldReturn := TRUE;
                    CommandAck := FALSE;
                    MessagePackerFb.PackKvStr(ADR('err'), ADR('flyevent_reject'));
                    GVL.FlyEventRejectNakCount := GVL.FlyEventRejectNakCount + 1;
                END_IF;
                GVL.minfo_buf_ridx.ConsumeTail();
            ELSE
                // R11 fix: same full-queue wedge as the M4 branch above.
                ShouldReturn := TRUE;
                CommandAck := FALSE;
                MessagePackerFb.PackKvStr(ADR('err'), ADR('flyevent_buffer_full'));
                GVL.FlyEventBufferFullNakCount := GVL.FlyEventBufferFullNakCount + 1;
                GVL.minfo_buf_ridx.ConsumeTail();
            END_IF;

        ELSIF (CommandType = 'G1') THEN
            // PH#6: dedupe scan. UI-side retry on TCP jitter or a double-
            // click can re-send the same G1 with the same CommandId. If
            // we already accepted that CommandId recently, replay the
            // cached movement_id with dedup:TRUE and skip the actual
            // MoveLinearAbsoluteFb.Execute=1 -- otherwise we'd queue two
            // physical moves for one logical request. CommandId=0 is the
            // no-id sentinel and never matches.
            DupeMatchIdx := -1;
            IF (CommandId <> 0) THEN
                FOR DupeLoopIdx := 0 TO DUPE_RING_SIZE - 1 DO
                    IF (RecentCmdIds[DupeLoopIdx] = CommandId) THEN
                        DupeMatchIdx := DupeLoopIdx;
                        EXIT;
                    END_IF;
                END_FOR;
            END_IF;

            IF (DupeMatchIdx >= 0) THEN
                MessagePackerFb.PackKvLint(ADR('movement_id'), TO_LINT(RecentCmdMoveIds[DupeMatchIdx]));
                MessagePackerFb.PackKvBool(ADR('dedup'), TRUE);
                ShouldReturn := TRUE;
                CommandAck := TRUE;
                GVL.DupeCommandCount := GVL.DupeCommandCount + 1;
                GVL.minfo_buf_ridx.ConsumeTail();

            // Coord-system gate. The PLC applies the machine frame itself
            // on Ready entry (CheckAxisGroupReady); SetCoord0/1 also set
            // it. Refuse G1 until one of them has since the last UnInited
            // / Error entry, and check the group's actual transform.
            ELSIF (NOT GVL.CoordSystemConfigured) THEN
                MessagePackerFb.PackKvStr(ADR('err'), ADR('coord_not_configured'));
                GVL.CoordNotConfiguredNakCount := GVL.CoordNotConfiguredNakCount + 1;
                ShouldReturn := TRUE;
                CommandAck := FALSE;
                GVL.minfo_buf_ridx.ConsumeTail();

            // The transform being applied (SetCoord or the Ready-entry
            // auto-apply): hold the G1 until the group has it.
            ELSIF (NOT CoordFrameOk AND (ApplyCoordTransform OR SetCoordTransformFb.Busy)) THEN
                RetryMotionCommandCooldown := RETRY_COOLDOWN_G1_MS;

            // The group's actual transform is not the one set: never move
            // in an unknown frame.
            ELSIF (NOT CoordFrameOk) THEN
                MessagePackerFb.PackKvStr(ADR('err'), ADR('coord_mismatch'));
                GVL.CoordMismatchNakCount := GVL.CoordMismatchNakCount + 1;
                ShouldReturn := TRUE;
                CommandAck := FALSE;
                GVL.minfo_buf_ridx.ConsumeTail();
            ELSE
            // Phase 3: read `frame` FIRST so we can NAK before mutating
            // persistent MotionPose / Latest* modal state. A NAK that
            // happens after the unpacks (the prior shape of this code)
            // poisoned the "previous XYZ / F / ACC" defaults that
            // subsequent omit-field G1s rely on.
            G1FrameTag := TO_INT(MessageUnpackerFb.TryReadINT64('frame', 0));
            IF (G1FrameTag <> 0 AND G1FrameTag <> 1) THEN
                MessagePackerFb.PackKvStr(ADR('err'), ADR('bad_frame'));
                GVL.Coord1BadFrameNakCount := GVL.Coord1BadFrameNakCount + 1;
                ShouldReturn := TRUE;
                CommandAck := FALSE;
                GVL.minfo_buf_ridx.ConsumeTail();
            ELSIF (G1FrameTag = 1 AND NOT GVL.Coord1Bound) THEN
                MessagePackerFb.PackKvStr(ADR('err'), ADR('coord1_not_bound'));
                GVL.Coord1NotBoundNakCount := GVL.Coord1NotBoundNakCount + 1;
                ShouldReturn := TRUE;
                CommandAck := FALSE;
                GVL.minfo_buf_ridx.ConsumeTail();
            ELSE
            MotionPose.c.X := MessageUnpackerFb.TryReadREAL('X', MotionPose.c.X);
            MotionPose.c.Y := MessageUnpackerFb.TryReadREAL('Y', MotionPose.c.Y);
            MotionPose.c.Z := MessageUnpackerFb.TryReadREAL('Z', MotionPose.c.Z);
            // A: degrees -> Kin_CAxis pose units (/10 wrap), on the fixed
            // zero A_AXIS_ZERO_DEG, with the frame's A rotation cancelled
            // (the planner subtracts CoordTransform.A from the pose A).
            // Constants and the why: AxisGroupSM VAR CONSTANT.
            MotionPoseTempReal := MessageUnpackerFb.TryReadREAL('A', G1_A_UNSET_SENTINEL);
            IF (MotionPoseTempReal <> G1_A_UNSET_SENTINEL) THEN
                G1ADeg := MotionPoseTempReal;
            END_IF;
            MotionPose.c.A := (G1ADeg + A_AXIS_ZERO_DEG) / A_AXIS_KIN_WRAP_SCALE + CoordTransform.A;

            LatestFeedRate := MessageUnpackerFb.TryReadREAL('F', LatestFeedRate);
            LatestAcceleration := MessageUnpackerFb.TryReadREAL('ACC', LatestAcceleration);
            LatestDeceleration := MessageUnpackerFb.TryReadREAL('DEA', LatestDeceleration);
            LatestJerk := MessageUnpackerFb.TryReadREAL('JERK', LatestJerk);
            LatestFactor := MessageUnpackerFb.TryReadREAL('FAC', LatestFactor);
            IF (LatestFactor > 1) THEN LatestFactor := 1; END_IF;
            IF (LatestFactor < 0.001) THEN LatestFactor := 0.001; END_IF;

            CornerTransition := MessageUnpackerFb.TryReadREAL('Cor', CornerTransition);
            TransitionParameter[0] := CornerTransition;
            G1AbortMode := MessageUnpackerFb.TryReadBool('abort', FALSE);

            // Phase 4 step 2: frame=1 simply switches CoordSystem to
            // PCS_1. MC_TrackConveyorBelt keeps PCS_1 origin synced to
            // the belt every scan, so MotionPose is interpreted as the
            // tracking-frame target and the kernel handles the
            // synchronized handover during the move (the prior
            // hand-rolled "Coord1OriginNow add at MC call time" was a
            // frozen-target approximation -- replaced by SM3 native FB).
            G1TargetPose := MotionPose;
            IF (G1FrameTag = 1) THEN
                G1CoordSystem := SMC_COORD_SYSTEM.PCS_1;
            ELSE
                G1CoordSystem := SMC_COORD_SYSTEM.WCS;
            END_IF;

            MoveLinearAbsoluteFb(
                AxisGroup := AxisGroupManagerFb._agAxisGroup,
                Execute := 1,
                Position := G1TargetPose,
                Velocity := LatestFeedRate * OverrideNow,
                // speed override (GVL.OverrideFactor, see AxisGroupSM):
                // velocity x f, acceleration x f^2, jerk x f^3
                Acceleration := LatestAcceleration * OverrideNow * OverrideNow,
                Deceleration := LatestDeceleration * OverrideNow * OverrideNow,
                Jerk := LatestJerk * OverrideNow * OverrideNow * OverrideNow,
                CoordSystem := G1CoordSystem,
                BufferMode := SEL(G1AbortMode,
                    SEL(CornerTransition >= 1, SM3_Common.MC_BUFFER_MODE.Buffered, SM3_Common.MC_BUFFER_MODE.BlendingNext),
                    SM3_Common.MC_BUFFER_MODE.Aborting),
                TransitionMode := SM3_Robotics.MC_TRANSITION_MODE.TMCornerDistance,
                TransitionParameter := TransitionParameter,
                VelFactor := LatestFactor,
                AccFactor := LatestFactor,
                JerkFactor := LatestFactor,
                TorqueFactor := 1,
                Done => ,
                Busy => ,
                Active => ,
                MovementId =>
            );

            IF (MoveLinearAbsoluteFb.CommandAccepted) THEN
                GVL.minfo_buf_ridx.ConsumeTail();

                MessagePackerFb.PackKvLint(ADR('movement_id'), TO_LINT(MoveLinearAbsoluteFb.MovementId));

                // PH#6: record this accepted G1 in the dedupe ring so a
                // retransmit with the same CommandId hits the cache and
                // replays the movement_id instead of executing again.
                // Skip the no-id sentinel (CommandId=0) -- caching it
                // would collide every legacy/no-id G1 with each other.
                IF (CommandId <> 0) THEN
                    RecentCmdIds[RecentCmdRingHead] := CommandId;
                    RecentCmdMoveIds[RecentCmdRingHead] := MoveLinearAbsoluteFb.MovementId;
                    RecentCmdRingHead := (RecentCmdRingHead + 1) MOD DUPE_RING_SIZE;
                END_IF;

                ShouldReturn := TRUE;
                CommandAck := TRUE;
            ELSE
                RetryMotionCommandCooldown := RETRY_COOLDOWN_G1_MS;
                GVL.G1RetryCount := GVL.G1RetryCount + 1;
            END_IF;
            END_IF; // frame validation / MoveLinear
            END_IF; // dedupe / coord-gate / execute

        ELSIF (CommandType = 'getDigitalInputFlipCount') THEN

            MessagePackerFb.PackKvDint(ADR('raw'), TO_DINT(DigitalInputBits_Curr));

            MessagePackerFb.PackKvArray(ADR('fc'), 16);
            FOR StageLoopIdx := 0 TO 15 DO
                MessagePackerFb.PackElemDint(TO_DINT(DigitalInputFlipCounts[StageLoopIdx]));
            END_FOR;

            ShouldReturn := TRUE;
            CommandAck := TRUE;
            GVL.minfo_buf_ridx.ConsumeTail();

        ELSE
            // R2 fix: unknown motion cmd used to NAK bare (no err, no
            // counter) -- host saw ack:false with zero diagnosis.
            MessagePackerFb.PackKvStr(ADR('err'), ADR('unknown_cmd'));
            GVL.UnknownCmdNakCount := GVL.UnknownCmdNakCount + 1;
            GVL.minfo_buf_ridx.ConsumeTail();
            ShouldReturn := TRUE;
        END_IF;

        IF ShouldReturn = TRUE AND CommandId <> 0 THEN
            MessagePackerFb.PackKvDint(ADR('id'), CommandId);

            MessagePackerFb.PackKvBool(ADR('ack'), CommandAck);

            // Only commit the slot if we actually reserved one above
            // (SlotAvailable=FALSE: the pack wrote to the scratch slot) and
            // Wrapup produced a valid packet (see CommitReplySlotAck).
            IF MsgPakInfoWrapup(ResponsePacketPointer^) AND SlotAvailable THEN
                GVL.reMP_info_ridx.PushHead();
            END_IF;
        END_IF;
    END_IF;

(* ---- TickTtl.st ---- *)
METHOD TickTtl : BOOL
VAR_INPUT
    p : POINTER TO FlyEventData;
END_VAR
(* =========== IMPLEMENTATION =========== *)
// Common TTL-decrement-and-expire logic factored out of
// ProcessFlyEventsAndIo. Each of DistanceTrigger / MovmentProgress /
// PulseTrigger ran the same 7 lines verbatim in their ELSE branch.
//
// Returns TRUE when the TTL just expired (caller should set
// TriggerErrorCode = TRIGGER_TIMEOUT_ERR and run the trigger-fired
// path with the error). TimeToLiveMs = -1 means "no expiry"; only
// strictly positive values decay.
TickTtl := FALSE;
IF (p^.TimeToLiveMs > 0) THEN
    p^.TimeToLiveMs := p^.TimeToLiveMs - BusPeriod;
    IF (p^.TimeToLiveMs <= 0) THEN
        TickTtl := TRUE;
    END_IF;
END_IF;

(* ---- TryAcquireReplySlot.st ---- *)
METHOD TryAcquireReplySlot : BOOL
VAR_INPUT
    pDropClassCounter : POINTER TO UDINT;
END_VAR
(* =========== IMPLEMENTATION =========== *)
// Reply / event slot acquisition. Returns TRUE if a free reMP_info
// slot was reserved (caller may proceed to pack + CommitReplySlot*),
// FALSE if the ring is full (caller skips the pack body; drop counter
// already bumped here).
//
// On success: ResponsePacketPointer points at the reserved slot,
// MsgPakInfoClear has been called (ele_count = 0, whead = buf base),
// caller goes straight to PackKv* / PackKvMap etc.
//
// On full-ring failure: GVL.ReMpDropCount + the class-specific counter
// (pDropClassCounter, e.g. ADR(GVL.ReMpDropCount_TriggerEvent)) are
// both incremented. Pass 0 if no class-specific counter applies.
//
// Producer-only -- caller MUST NOT call .ConsumeTail on the reply ring.
// Pairs with CommitReplySlotAck (request reply) or CommitReplySlotEvent
// (unsolicited push event).
IF (GVL.reMP_info_ridx.Space() > 0) THEN
    ResponsePacketPointer := ADR(GVL.reMP_info_arr[GVL.reMP_info_ridx.GetHead()]);
    MsgPakInfoClear(ResponsePacketPointer^);
    MessagePackerFb.BindSlot(ResponsePacketPointer);  // builder pattern: pack helpers target this slot
    TryAcquireReplySlot := TRUE;
ELSE
    GVL.ReMpDropCount := GVL.ReMpDropCount + 1;
    IF pDropClassCounter <> 0 THEN
        pDropClassCounter^ := pDropClassCounter^ + 1;
    END_IF;
    TryAcquireReplySlot := FALSE;
END_IF;

(* ---- TryAcquireReplySlotOrScratch.st ---- *)
METHOD TryAcquireReplySlotOrScratch : BOOL
VAR_INPUT
    pDropClassCounter : POINTER TO UDINT;
END_VAR
(* =========== IMPLEMENTATION =========== *)
// Main-dispatcher slot acquisition with scratch fallback. Always
// succeeds at giving the caller a slot to pack into -- if the real
// ring is full it routes the pack into GVL.reMP_info_scratch so the
// long ELSIF dispatch chain in DrainHostPackets can stay unchanged.
//
// Sets SlotAvailable as the return value:
//   TRUE  -> real slot reserved, CommitReplySlotOrScratch will PushHead
//   FALSE -> packed into scratch; CommitReplySlotOrScratch will NOT
//            PushHead (would corrupt a slot a consumer is reading)
//            and will bump the class-specific drop counter.
//
// pDropClassCounter is bumped IN CommitReplySlotOrScratch on the FALSE
// branch (not here) so callers that bail out before commit don't get
// counted.
IF (GVL.reMP_info_ridx.Space() > 0) THEN
    SlotAvailable := TRUE;
    ResponsePacketPointer := ADR(GVL.reMP_info_arr[GVL.reMP_info_ridx.GetHead()]);
ELSE
    SlotAvailable := FALSE;
    ResponsePacketPointer := ADR(GVL.reMP_info_scratch);
END_IF;
MsgPakInfoClear(ResponsePacketPointer^);
MessagePackerFb.BindSlot(ResponsePacketPointer);  // builder pattern: pack helpers target this slot (real OR scratch)
TryAcquireReplySlotOrScratch := SlotAvailable;

(* ---- UpdateDiWatch.st ---- *)
METHOD UpdateDiWatch : BOOL
VAR
    i       : INT;
    bitNow  : BOOL;
    bitPrev : BOOL;
    sent    : INT;
END_VAR
(* =========== IMPLEMENTATION =========== *)
// Digital-input change events (SYS DI_WATCH): the host registers pins, an
// edge filter and a throttle; every scan (1 ms) this tracks each watched
// pin and pushes {kind:'event', name:'DI'} when it changes. The first
// matching edge after a quiet throttle period goes out at once; changes
// inside the throttle window are summarised into one event at its end,
// so nothing is lost to the throttle:
//   state        level now
//   flips        changes since the last event (any edge)
//   high_ms      time high since the last event
//   max_high_ms / max_low_ms   longest run at each level that ended since the
//                last event, or is still going (a run is not cut by an event)
//   t_first      RuntimeMs of the first change since the last event
//   reel_odo_um  reel odometer (GVL.ReelOdoMm, um) at that first change
//   t            RuntimeMs now
// A full reply ring defers the push to a later scan (at most 2 per scan,
// and never into the last 2 slots, which stay for command replies).
// Generic on purpose: what an input means is the host's business.
IF NOT DiWatchInit THEN
    DiWatchPrev := DigitalInputBits_Curr;
    DiWatchInit := TRUE;
END_IF;
IF NOT TCP_MSGPAK_Server.fbMyServer.CLIENT.xActive THEN
    // host gone: nobody to tell; it registers again when it reconnects
    DiWatchMask := 0;
END_IF;
IF DiWatchMask = 0 THEN
    DiWatchPrev := DigitalInputBits_Curr;
    RETURN;
END_IF;
sent := 0;
FOR i := 0 TO 15 DO
    IF (SHR(DiWatchMask, i) AND 1) <> 0 THEN
        bitNow  := (SHR(DigitalInputBits_Curr, i) AND 1) <> 0;
        bitPrev := (SHR(DiWatchPrev, i) AND 1) <> 0;
        IF bitNow <> bitPrev THEN
            // close the run of the level just left
            IF bitPrev THEN
                DiWMaxHighMs[i] := MAX(DiWMaxHighMs[i], DiWRunMs[i]);
            ELSE
                DiWMaxLowMs[i] := MAX(DiWMaxLowMs[i], DiWRunMs[i]);
            END_IF;
            DiWRunMs[i] := 0;
            IF DiWFlips[i] = 0 THEN
                DiWFirstMs[i] := RuntimeMs;
                DiWReelOdo[i] := GVL.ReelOdoMm;
            END_IF;
            DiWFlips[i] := DiWFlips[i] + 1;
            IF (bitNow AND ((SHR(DiWatchRise, i) AND 1) <> 0))
               OR (NOT bitNow AND ((SHR(DiWatchFall, i) AND 1) <> 0)) THEN
                DiWPending[i] := TRUE;
            END_IF;
        END_IF;
        DiWRunMs[i] := DiWRunMs[i] + TO_DINT(BusPeriod);
        IF bitNow THEN
            DiWHighMs[i] := DiWHighMs[i] + TO_DINT(BusPeriod);
        END_IF;
        IF DiWPending[i] AND (sent < 2)
           AND ((RuntimeMs - DiWLastSentMs[i]) >= DiWatchThrottleMs[i])
           AND (GVL.reMP_info_ridx.Space() > 2) THEN
            IF TryAcquireReplySlot(0) THEN
                MessagePackerFb.PackKvStr(ADR('kind'), ADR('event'));
                MessagePackerFb.PackKvStr(ADR('name'), ADR('DI'));
                MessagePackerFb.PackKvDint(ADR('pin'), i);
                MessagePackerFb.PackKvBool(ADR('state'), bitNow);
                MessagePackerFb.PackKvLint(ADR('flips'), UDINT_TO_LINT(DiWFlips[i]));
                MessagePackerFb.PackKvDint(ADR('high_ms'), DiWHighMs[i]);
                IF bitNow THEN
                    MessagePackerFb.PackKvDint(ADR('max_high_ms'), MAX(DiWMaxHighMs[i], DiWRunMs[i]));
                    MessagePackerFb.PackKvDint(ADR('max_low_ms'), DiWMaxLowMs[i]);
                ELSE
                    MessagePackerFb.PackKvDint(ADR('max_high_ms'), DiWMaxHighMs[i]);
                    MessagePackerFb.PackKvDint(ADR('max_low_ms'), MAX(DiWMaxLowMs[i], DiWRunMs[i]));
                END_IF;
                MessagePackerFb.PackKvLint(ADR('t_first'), DiWFirstMs[i]);
                MessagePackerFb.PackKvLint(ADR('reel_odo_um'), LREAL_TO_LINT(DiWReelOdo[i] * 1000.0));
                MessagePackerFb.PackKvLint(ADR('t'), RuntimeMs);
                CommitReplySlotEvent();
                DiWFlips[i] := 0;
                DiWHighMs[i] := 0;
                DiWMaxHighMs[i] := 0;
                DiWMaxLowMs[i] := 0;
                DiWPending[i] := FALSE;
                DiWLastSentMs[i] := RuntimeMs;
                GVL.DiEventCount := GVL.DiEventCount + 1;
                sent := sent + 1;
            END_IF;
        END_IF;
    END_IF;
END_FOR;
DiWatchPrev := DigitalInputBits_Curr;

(* ---- UpdateMotionProgress.st ---- *)
(* =========== IMPLEMENTATION =========== *)
TempMovementId := GroupReadPositionFb.MovementId;
// If either MC read FB is in error, don't propagate its outputs -- they
// may be stale. Freeze buffer size to 0 so ProcessMotionPacket won't
// treat "buffer has room" as "motion is healthy" and accept a new
// move on top of an errored group.
IF GroupReadStatusFb.Error OR GroupReadPositionFb.Error THEN
    MotionBufferSize := 0;
ELSIF (GroupReadPositionFb.MovementId = 0) THEN
    MotionBufferSize := 0;
    CurrentMovementId := GroupReadStatusFb.LastAcceptedMovementId;
    CurrentMovementIdProgress := 1;
    IF (CurrentMovementId = 0) THEN
        CurrentMovementIdProgress := 0;
    END_IF;
ELSE
    // Guard against underflow: both are unsigned SMC_Movement_Id.
    // LastAccepted < current shouldn't happen, but could during
    // a reset race. Clamp to 0 rather than wrapping to huge ULINT.
    IF GroupReadStatusFb.LastAcceptedMovementId >= GroupReadPositionFb.MovementId THEN
        MotionBufferSize := GroupReadStatusFb.LastAcceptedMovementId - GroupReadPositionFb.MovementId;
    ELSE
        MotionBufferSize := 0;
    END_IF;

    IF (CurrentMovementId <> GroupReadPositionFb.MovementId) THEN
        CurrentMovementId := GroupReadPositionFb.MovementId;
    END_IF;

    CurrentMovementIdProgress := GroupReadPositionFb.Position;
END_IF;

IF (CurrentMovementId <> PrevMotionStateId OR CurrentMovementIdProgress <> PrevMotionStateProgress) THEN
    MotionStateString := CONCAT(
        CONCAT(TO_STRING(CurrentMovementId), ' '),
        TO_STRING(CurrentMovementIdProgress)
    );
    PrevMotionStateId := CurrentMovementId;
    PrevMotionStateProgress := CurrentMovementIdProgress;
END_IF;

// MOVE_DONE push event: MotionBufferSize transition >0 -> 0 with a
// non-zero LastAcceptedMovementId means the queued motion drained.
// The UI can gate "ready for next step" on this event instead of
// polling movement_id via GET_MACHINE_STATE at high frequency.
// Envelope matches ST_CHG: kind='event', name='MOVE_DONE'.
//
// PH#5: edge-detection latches PendingMoveDoneId. A separate retry
// block below tries to push every scan until the ring has space, so
// a transient ring-full doesn't lose the event (UI would otherwise
// wait up to 1s for the GET_MACHINE_STATE poll to notice).
// R10 fix (test_plc_refactor_findings): the >0 -> 0 edge also fires when
// an error/abort FLUSHES the buffer (error freeze above forces
// MotionBufferSize:=0; GroupStop drops MovementId to 0) -- that is not a
// completion. Latching it emitted MOVE_DONE for an aborted move and
// advanced last_completed_movement_id past moves that never ran, which
// the §4(2) resume reconcile reads as "intent completed" -> skipped
// blow-off -> double reel advance. Only latch the edge while the group
// is genuinely healthy and in Ready; an abort path must leave
// PrevCompletedMovementId at the last move that truly finished.
IF (PrevMotionBufferSizeForEvent > 0
    AND MotionBufferSize = 0
    AND GroupReadStatusFb.LastAcceptedMovementId <> 0
    AND GroupReadStatusFb.LastAcceptedMovementId <> PrevCompletedMovementId
    AND AxisGroupManagerFb._eState = E_RobotState.Ready
    AND NOT GroupReadStatusFb.Error
    AND NOT GroupReadPositionFb.Error
    AND NOT GroupReadStatusFb.GroupErrorStop) THEN
    // Newest edge wins: if a previous MOVE_DONE was pending and a new
    // movement just completed before we got to push it, just publish
    // the newer one. UI watches for movement_id gaps and surfaces the
    // skip; losing the older intermediate event is acceptable.
    PendingMoveDoneId := GroupReadStatusFb.LastAcceptedMovementId;
END_IF;
PrevMotionBufferSizeForEvent := MotionBufferSize;

// Retry pump: try until the ring has space. Producer-only on
// reMP_info_ridx -- never ConsumeTail here.
IF PendingMoveDoneId <> 0 THEN
    // Retry-style emit: use ProbeReplySlot (no per-scan drop-counter
    // bump). Only the final give-up below bumps the class-specific
    // PendingMoveDoneDropCount once.
    IF ProbeReplySlot() THEN
        MessagePackerFb.PackKvStr(ADR('kind'), ADR('event'));
        MessagePackerFb.PackKvStr(ADR('name'), ADR('MOVE_DONE'));
        MessagePackerFb.PackKvLint(ADR('movement_id'), TO_LINT(PendingMoveDoneId));
        MessagePackerFb.PackKvLint(ADR('runtime_ms'), RuntimeMs);
        CommitReplySlotEvent();
        PrevCompletedMovementId := PendingMoveDoneId;
        PendingMoveDoneId := 0;
        PendingMoveDoneRetryScans := 0;
    ELSE
        // Audit-fix: ring permanently full -> drop and move on. Without
        // this, a stuck consumer would leave PendingMoveDoneId asserted
        // forever and silently swallow every subsequent MOVE_DONE edge
        // (newest-wins overwrites the latch each scan; the UI has no
        // way to know it's stuck).
        //
        // PR review fix: drop ONLY the pending event; do NOT advance
        // PrevCompletedMovementId here. PrevCompletedMovementId is the
        // host-visible last_completed_movement_id used by the §4(2)
        // resume reconcile (scratchpad intent_movement_id vs this
        // field). Advancing it without successfully delivering MOVE_DONE
        // would tell the host "the move that you have an intent for
        // already completed" when in fact the host never saw the event.
        // Worst-case result: renderer skips a blow_off and reel
        // double-advances.
        PendingMoveDoneRetryScans := PendingMoveDoneRetryScans + 1;
        IF PendingMoveDoneRetryScans >= PENDING_RETRY_MAX_SCANS THEN
            PendingMoveDoneId := 0;
            PendingMoveDoneRetryScans := 0;
            GVL.PendingMoveDoneDropCount := GVL.PendingMoveDoneDropCount + 1;
        END_IF;
    END_IF;
END_IF;

ShouldReturn := FALSE;
CommandAck := FALSE;

(* ---- UpdateRuntimeAndInputEvent.st ---- *)
(* =========== IMPLEMENTATION =========== *)
IF BusPeriodUs = 0 THEN
    BpH := CmpIecTask.IecTaskGetCurrent(ADR(BpR));
    IF BpR = 0 THEN
        BpP := CmpIecTask.IecTaskGetInfo3(BpH, ADR(BpR));
        IF (BpR = 0) AND (BpP <> 0) AND (BpP^.dwInterval >= 1000) THEN
            BusPeriodUs := BpP^.dwInterval;
            BusPeriod := DWORD_TO_DINT(BusPeriodUs / 1000);
            GVL.EcNominalUs := DWORD_TO_LREAL(BusPeriodUs);
        END_IF;
    END_IF;
END_IF;
RuntimeMs := RuntimeMs + BusPeriod;

// VisuEventControl=0 is the idle/no-op default so the TCP handler
// (ProcessSystemPacket below) can own InputEvent without being
// clobbered by this block on the next cycle. Visualisation buttons
// should write 1..6 momentarily and reset to 0.
CASE VisuEventControl OF
    1: InputEvent := E_RobotEvent.EV_POWER_ON;
    2: InputEvent := E_RobotEvent.EV_GROUP_ENABLE;
    3: InputEvent := E_RobotEvent.EV_HOME_GO;
    4: InputEvent := E_RobotEvent.EV_ERROR;
    5: InputEvent := E_RobotEvent.EV_RESET;
    6: InputEvent := E_RobotEvent.EV_HOME_GO_FORCE_SKIP;
END_CASE;

IF (PreviousInputEvent <> InputEvent) THEN
    AxisGroupManagerFb.TRANSITION(
        eEvent := InputEvent
    );
END_IF;

PreviousInputEvent := InputEvent;
IF TO_INT(AxisGroupManagerFb._eState) <> PrevAxisGroupState THEN
    StateString := TO_STRING(AxisGroupManagerFb._eState);
    // PH#8: latch "from" for the deferred ST_CHG emit instead of pushing
    // inline. The retry pump below tries every scan until the ring has
    // space, so a transient ring-full no longer drops the event. Skip
    // PrevAxisGroupState=-1 (cold-boot sentinel, no "from" to report).
    // Newest-edge-wins: rapid A->B->C while pending overwrites "from"
    // each edge -- UI sees ST_CHG{from=B,to=C}+seq gap and reconciles.
    IF (PrevAxisGroupState >= 0) THEN
        PendingStChgFromState := TO_DINT(PrevAxisGroupState);
    END_IF;
    // Audit-fix: clear the G1 dedupe ring on entry to Error or UnInited.
    // The (CommandId, MovementId) pairs are scoped to the in-flight session;
    // after a fault or full reset the cached MovementIds correspond to
    // motions that no longer exist. If UI restarts (CommandId counter
    // resets to 0) or a deterministic id-from-cmd-name scheme is used, an
    // unscrubbed ring would replay a stale MovementId on the next G1 with
    // a colliding CommandId -- silent no-op from the operator's view, or
    // worse, the wrong motion appearing to "succeed".
    IF (AxisGroupManagerFb._eState = E_RobotState.Error
        OR AxisGroupManagerFb._eState = E_RobotState.UnInited) THEN
        FOR DupeLoopIdx := 0 TO DUPE_RING_SIZE - 1 DO
            RecentCmdIds[DupeLoopIdx] := 0;
            RecentCmdMoveIds[DupeLoopIdx] := 0;
        END_FOR;
        RecentCmdRingHead := 0;
        // Fly events belong to the run that just faulted (FlushFlyEvents
        // answers / reports / finishes them instead of dropping silently).
        FlushFlyEvents(notify := TCP_MSGPAK_Server.fbMyServer.CLIENT.xActive);
    END_IF;

    PrevAxisGroupState := TO_INT(AxisGroupManagerFb._eState);
END_IF;

// The host went away: what it queued belongs to its session. An M4 aimed
// at "the next move" would otherwise fire on the new session's first G1,
// and the duplicate filter would match the new session's restarted ids.
// Packets it sent that are not processed yet are dropped too (nobody to
// answer; an M4 registered after the flush would be an orphan). Motion
// the group already accepted runs to its end.
IF PrevClientActive AND NOT TCP_MSGPAK_Server.fbMyServer.CLIENT.xActive THEN
    FOR DupeLoopIdx := 0 TO DUPE_RING_SIZE - 1 DO
        RecentCmdIds[DupeLoopIdx] := 0;
        RecentCmdMoveIds[DupeLoopIdx] := 0;
    END_FOR;
    RecentCmdRingHead := 0;
    // Consumer side of both SPSC rings (the Comm task only pushes).
    WHILE GVL.minfo_buf_ridx.Size() > 0 DO
        GVL.minfo_buf_ridx.ConsumeTail();
        GVL.HostGonePacketDropCount := GVL.HostGonePacketDropCount + 1;
    END_WHILE;
    WHILE GVL.sysinfo_buf_ridx.Size() > 0 DO
        GVL.sysinfo_buf_ridx.ConsumeTail();
        GVL.HostGonePacketDropCount := GVL.HostGonePacketDropCount + 1;
    END_WHILE;
    RetryMotionCommandCooldown := 0;
    FlushFlyEvents(notify := FALSE);
END_IF;
PrevClientActive := TCP_MSGPAK_Server.fbMyServer.CLIENT.xActive;

// ST_CHG retry pump (PH#8). PendingStChgFromState >= 0 means an edge is
// waiting to publish; "to" is the current _eState at retry time, which
// under newest-wins always pairs cleanly with the latched "from".
// Producer-only on reMP_info_ridx -- never ConsumeTail here. No drop
// counter bump: ring-full just means "try again next scan", not loss.
IF (PendingStChgFromState >= 0) THEN
    IF ProbeReplySlot() THEN
        StateString := TO_STRING(AxisGroupManagerFb._eState);
        MessagePackerFb.PackKvStr(ADR('kind'), ADR('event'));
        MessagePackerFb.PackKvStr(ADR('name'), ADR('ST_CHG'));
        MessagePackerFb.PackKvDint(ADR('st'), AxisGroupManagerFb._eState);
        MessagePackerFb.PackKvStr(ADR('st_str'), ADR(StateString));
        MessagePackerFb.PackKvDint(ADR('from'), PendingStChgFromState);
        MessagePackerFb.PackKvLint(ADR('runtime_ms'), RuntimeMs);
        CommitReplySlotEvent();
        GVL.StateChangeEventCount := GVL.StateChangeEventCount + 1;
        PendingStChgFromState := -1;
        PendingStChgRetryScans := 0;
    ELSE
        // Bound the retry. Drop after PENDING_RETRY_MAX_SCANS so a
        // permanently-stuck ring doesn't swallow every subsequent
        // ST_CHG edge silently. Newest-wins means the latched "from"
        // would otherwise just keep getting overwritten while never
        // landing.
        PendingStChgRetryScans := PendingStChgRetryScans + 1;
        IF PendingStChgRetryScans >= PENDING_RETRY_MAX_SCANS THEN
            PendingStChgFromState := -1;
            PendingStChgRetryScans := 0;
            GVL.PendingStChgDropCount := GVL.PendingStChgDropCount + 1;
        END_IF;
    END_IF;
END_IF;

// COORD_SET push event: edge-detect on GVL.CoordSystemConfigured (both
// directions). UnInited entry clears the gate; SetCoord0/1 raises it.
// The falling edge matters as much as the rising one -- after a reset
// the operator's first G1 will NAK with err='coord_not_configured'
// unless they reconfigure, so the UI needs to know the gate dropped
// without polling GET_MACHINE_STATE.
// Envelope matches ST_CHG: kind='event', name='COORD_SET', plus a BOOL
// `value` carrying the new gate state.
IF (GVL.CoordSystemConfigured <> PrevCoordSet) THEN
    // Drop-newest on overflow (see UpdateMotionProgress for rationale).
    IF TryAcquireReplySlot(ADR(GVL.ReMpDropCount_CoordSet)) THEN
        MessagePackerFb.PackKvStr(ADR('kind'), ADR('event'));
        MessagePackerFb.PackKvStr(ADR('name'), ADR('COORD_SET'));
        MessagePackerFb.PackKvBool(ADR('value'), GVL.CoordSystemConfigured);
        MessagePackerFb.PackKvLint(ADR('runtime_ms'), RuntimeMs);
        CommitReplySlotEvent();
    END_IF;
END_IF;
PrevCoordSet := GVL.CoordSystemConfigured;

// HEARTBEAT push event. Periodic (HEARTBEAT_INTERVAL_MS, default 500) so
// the UI can detect a dead PLC socket without sending SYS/PING -- and so
// it has a regular cadence to anchor seq-gap detection (if no other event
// fires for seconds, an "expected next seq" still progresses every 500ms).
// Drop-newest on overflow: ring full means the UI has bigger problems
// than a missing heartbeat tick; ReMpDropCount grows and the seq jumps.
IF (LastHeartbeatMs = 0) OR (RuntimeMs - LastHeartbeatMs >= HEARTBEAT_INTERVAL_MS) THEN
    IF TryAcquireReplySlot(ADR(GVL.ReMpDropCount_Heartbeat)) THEN
        MessagePackerFb.PackKvStr(ADR('kind'), ADR('event'));
        MessagePackerFb.PackKvStr(ADR('name'), ADR('HEARTBEAT'));
        MessagePackerFb.PackKvLint(ADR('runtime_ms'), RuntimeMs);
        MessagePackerFb.PackKvLint(ADR('remp_drop_count'), TO_LINT(GVL.ReMpDropCount));
        // Per-type drop breakdown so DiagPanel can tell "lost replies" (real
        // problem) from "lost heartbeat tick" (cosmetic) without polling.
        MessagePackerFb.PackKvLint(ADR('drops_reply'),  TO_LINT(GVL.ReMpDropCount_Reply));
        MessagePackerFb.PackKvLint(ADR('drops_events'), TO_LINT(GVL.ReMpDropCount_StChg + GVL.ReMpDropCount_CoordSet + GVL.ReMpDropCount_Heartbeat + GVL.ReMpDropCount_TriggerEvent));
        CommitReplySlotEvent();
    END_IF;
    LastHeartbeatMs := RuntimeMs;
END_IF;
